// TIA Portal V16 export
// export: Created 2024-12-03T15:41:43.6424382Z, ExportSetting WithDefaults, DisplayName Totally Integrated Automation Portal, DisplayVersion V16 Update 6, DisplayName TIA Portal Version Control Interface, DisplayVersion V16 Update 2, DisplayName TIA Portal Openness, DisplayVersion V16 Update 6, DisplayName TIA Portal Teamcenter Gateway, DisplayVersion V16, DisplayName SINAMICS Startdrive Advanced, DisplayVersion V16 Update 5, DisplayName SINAMICS Startdrive G130, G150, S120, S150, SINAMICS MV, S210, DisplayVersion V16 Update 5, DisplayName SINAMICS Startdrive G110M, G120, G120C, G120D, G120P, G115D, DisplayVersion V16 Update 5, DisplayName STEP 7 Professional, DisplayVersion V16 Update 6, DisplayName STEP 7 Safety, DisplayVersion V16, DisplayName WinCC Advanced / Unified PC, DisplayVersion V16 Update 6
FUNCTION_BLOCK "EMG_STATUS_FB"   // FB10, SCL
{ S7_Optimized_Access := 'TRUE' }
VERSION : 0.1
// stored: AutoNumber true, IsIECCheckEnabled false, IsRetainMemResEnabled false, MemoryReserve 100, SetENOAutomatically false, UDAEnableTagReadback false
   VAR_INPUT
      I_BTTN_STATUS_OK : Bool;
      I_AlarmInfoBttnPressed : String[100];
      I_EMG_ACTIVATED : Bool;
      I_EmgName : String[100];
      I_UseBttnPressedALarm : Bool := true;
      I_UseEmgNotActiveAlarm : Bool := true;
   END_VAR
   VAR_OUTPUT
      O_AlarmActive : Bool;
   END_VAR
   VAR_IN_OUT
      IO_STATUS : "EMG_Status_UDT";
   END_VAR
   VAR
      alarmBTNNPRessed : Program_Alarm;
      alarmEmgNotActive : Program_Alarm;
   END_VAR
   VAR_TEMP
      T_ButtonActive : Bool;
      T_EmgActive : Bool;
   END_VAR
BEGIN
   REGION Check button is pressed

       #T_ButtonActive := NOT #I_BTTN_STATUS_OK AND #I_UseBttnPressedALarm;

       // #alarmBTNNPRessed(SIG:=#T_ButtonActive,
       //                   SD_2 := #I_AlarmInfoBttnPressed, SD_3 := #I_EmgName);

   END_REGION

   REGION Check button pressed and EMG nok

       #T_EmgActive := #I_BTTN_STATUS_OK AND NOT #I_EMG_ACTIVATED AND #I_UseEmgNotActiveAlarm;
       // #alarmEmgNotActive(SIG:=#T_EmgActive,
       //                    SD_1:=#I_EmgName);

   END_REGION

   REGION ALARM ACTIVE

       #O_AlarmActive := #T_ButtonActive OR #T_EmgActive;

   END_REGION

   REGION BUILD STATUS

       #IO_STATUS.emgNok := #T_ButtonActive OR #T_EmgActive;
       #IO_STATUS.activated := #T_ButtonActive;
       #IO_STATUS.waitingForReset := #T_EmgActive;

   END_REGION
END_FUNCTION_BLOCK
